TYPE ShutterConfigs :
STRUCT
	Ed12dssShutterConfig : Ed12dssShutterConfig;
	Sh10pilShutterConfig : Sh10pilShutterConfig;
END_STRUCT
END_TYPE

(* stored: Version 1.1.0.1, ProductVersion 3.1.4024.3
   DUT ShutterConfigs: Id {1f941dc3-8fed-44b4-9d2e-8fb33ae4e1d1} *)
